// TIA Portal V20 export
FUNCTION_BLOCK "LER_RFID"   // FB115, LAD
// stored: Access Published, MemoryReserve 100, SetENOAutomatically false
   VAR_INPUT
      enable : Bool;
      enableManualCmds : Bool;
      bobinChuck : Bool;
   END_VAR
   VAR_OUTPUT
      error : Bool;
      status : DWord;
   END_VAR
   VAR_IN_OUT
      RFID_Chanel : TO_IDENT;
      IdentRfAntena : "LSicar_typeIdentInterfaceHmi";
      moduleInterface : "LER_typeRFIDInterface";
   END_VAR
   VAR
      instResetReader : Reset_Reader;
      instRead : Read;
      instWrite : Write;
      instInventory : Inventory;
      statResetReaderUDT : "LER_typeResetReaderUDT";
      statReadUDT : "LER_typeReadWriteUDT";
      statWriteUDT : "LER_typeReadWriteUDT";
      statInventoryUDT : "LER_typeInventoryUDT";
      statResultRFIDReset : Bool;
      statPulse : Array[0..9] of Bool;
      statTonTimer : TON_TIME;
      statBobinData : IID_IN_I_81;
      statRFID_str : String[32];
      statEPCID_str : String[32];
      statHi : Byte;
      statLo : Byte;
      statHexArray : Array[0..15] of Char;
   END_VAR
   VAR_TEMP
      resultRFID_Delete : String;
      resultData_Delete : WString;
      resultid_Delete : SInt;
      tempRet_Val : Word;
      tempBobinEPCData : Array[1..62] of Byte;
      i : Int;
      HI : Int;
      LO : Int;
   END_VAR
   VAR CONSTANT
      FALSE : Bool;
      deviceType : WString := WSTRING#'RF680R';
      deviceId : SInt := 6;   // RF600 = 6
      tagType : WString := WSTRING#'RFID';
   END_VAR
   // statHexArray[0] := '0';
   // statHexArray[1] := '1';
   // statHexArray[2] := '2';
   // statHexArray[3] := '3';
   // statHexArray[4] := '4';
   // statHexArray[5] := '5';
   // statHexArray[6] := '6';
   // statHexArray[7] := '7';
   // statHexArray[8] := '8';
   // statHexArray[9] := '9';
   // statHexArray[10] := 'A';
   // statHexArray[11] := 'B';
   // statHexArray[12] := 'C';
   // statHexArray[13] := 'D';
   // statHexArray[14] := 'E';
   // statHexArray[15] := 'F';
   VAR_TEMP   // added for the SCL form of the ladder/FBD networks
      _w1 : Bool;
   END_VAR
BEGIN

REGION Network 1 (SCL): Input Mapping
   // READ
   #statReadUDT.Input.addrTag := #moduleInterface.configuration.addrTag;
   #statReadUDT.Input.lengthData := #moduleInterface.configuration.lengthData;

   // INVENTORY
   #statInventoryUDT.Input.attribute := #moduleInterface.configuration.attribute;
   #statInventoryUDT.Input.duration := #moduleInterface.configuration.duration;
   #statInventoryUDT.Input.durUnit := #moduleInterface.configuration.durUnit;

   IF #enableManualCmds OR true THEN
       #statResetReaderUDT.Input.execute := #moduleInterface.commands.ResetReq OR #IdentRfAntena.pushbutton.%X0;
       #statReadUDT.Input.execute := #moduleInterface.commands.readReq OR #IdentRfAntena.pushbutton.%X1;
       #statWriteUDT.Input.execute := #moduleInterface.commands.writeReq OR #IdentRfAntena.pushbutton.%X2;
       #statResultRFIDReset := #moduleInterface.commands.resultRFIDReset OR #IdentRfAntena.pushbutton.%X3;
       #statInventoryUDT.Input.execute := #moduleInterface.commands.inventoryReq OR #statReadUDT.Output.done;

   END_IF;
END_REGION

REGION Network 2: Reset Reader
   // The Reset block sets the reader to a operational state. The Reset also acknowledges error conditions of the reader and resets a reader from a falty state to a OK-state.
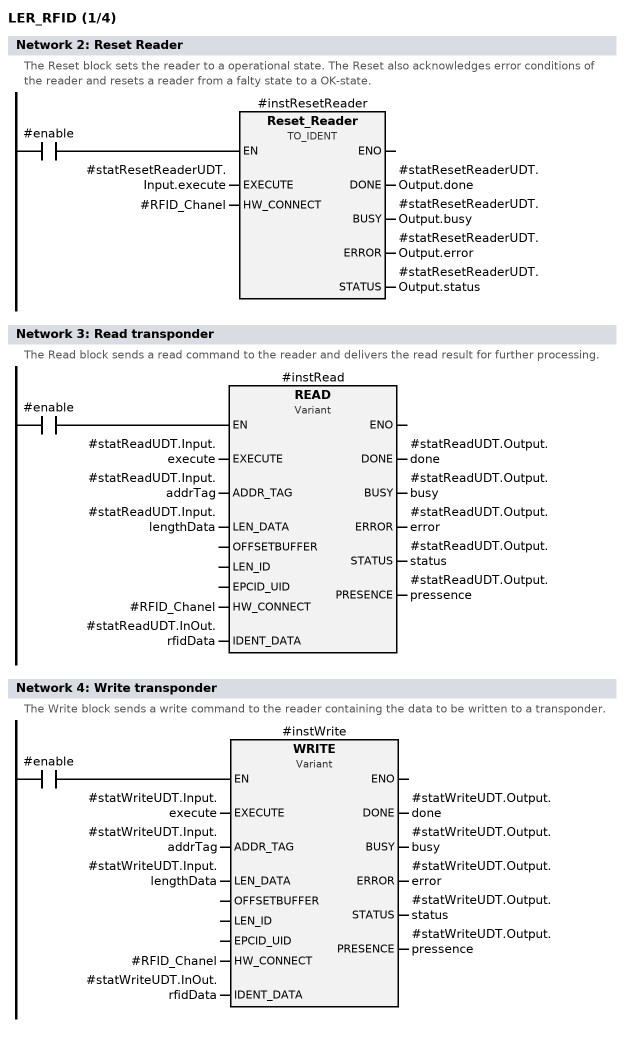
   RUNG wire#powerrail
      Contact( #enable )
      { S7_Templates := "connect_type := TO_IDENT" } #instResetReader.Reset_Reader(EXECUTE := #statResetReaderUDT.Input.execute, HW_CONNECT := #RFID_Chanel, DONE => #statResetReaderUDT.Output.done, BUSY => #statResetReaderUDT.Output.busy, ERROR => #statResetReaderUDT.Output.error, STATUS => #statResetReaderUDT.Output.status)
   END_RUNG
   // the same network as SCL:
   IF #enable THEN
       #instResetReader(EXECUTE := #statResetReaderUDT.Input.execute,   // Reset_Reader
                        HW_CONNECT := #RFID_Chanel,
                        DONE => #statResetReaderUDT.Output.done,
                        BUSY => #statResetReaderUDT.Output.busy,
                        ERROR => #statResetReaderUDT.Output.error,
                        STATUS => #statResetReaderUDT.Output.status);
   END_IF;
END_REGION

REGION Network 3: Read transponder
   // The Read block sends a read command to the reader and delivers the read result for further processing.
   RUNG wire#powerrail
      Contact( #enable )
      { S7_Templates := "[ident_data_type := Variant, connect_type := TO_IDENT]" } #instRead.Read(EXECUTE := #statReadUDT.Input.execute, ADDR_TAG := #statReadUDT.Input.addrTag, LEN_DATA := #statReadUDT.Input.lengthData, OFFSETBUFFER :=, LEN_ID :=, EPCID_UID :=, HW_CONNECT := #RFID_Chanel, IDENT_DATA := #statReadUDT.InOut.rfidData, DONE => #statReadUDT.Output.done, BUSY => #statReadUDT.Output.busy, ERROR => #statReadUDT.Output.error, STATUS => #statReadUDT.Output.status, PRESENCE => #statReadUDT.Output.pressence)
   END_RUNG
   // the same network as SCL:
   IF #enable THEN
       #instRead(EXECUTE := #statReadUDT.Input.execute,   // Read
                 ADDR_TAG := #statReadUDT.Input.addrTag,
                 LEN_DATA := #statReadUDT.Input.lengthData,
                 HW_CONNECT := #RFID_Chanel,
                 IDENT_DATA := #statReadUDT.InOut.rfidData,
                 DONE => #statReadUDT.Output.done,
                 BUSY => #statReadUDT.Output.busy,
                 ERROR => #statReadUDT.Output.error,
                 STATUS => #statReadUDT.Output.status,
                 PRESENCE => #statReadUDT.Output.pressence);
   END_IF;
END_REGION

REGION Network 4: Write transponder
   // The Write block sends a write command to the reader containing the data to be written to a transponder.
   RUNG wire#powerrail
      Contact( #enable )
      { S7_Templates := "[ident_data_type := Variant, connect_type := TO_IDENT]" } #instWrite.Write(EXECUTE := #statWriteUDT.Input.execute, ADDR_TAG := #statWriteUDT.Input.addrTag, LEN_DATA := #statWriteUDT.Input.lengthData, OFFSETBUFFER :=, LEN_ID :=, EPCID_UID :=, HW_CONNECT := #RFID_Chanel, IDENT_DATA := #statWriteUDT.InOut.rfidData, DONE => #statWriteUDT.Output.done, BUSY => #statWriteUDT.Output.busy, ERROR => #statWriteUDT.Output.error, STATUS => #statWriteUDT.Output.status, PRESENCE => #statWriteUDT.Output.pressence)
   END_RUNG
   // the same network as SCL:
   IF #enable THEN
       #instWrite(EXECUTE := #statWriteUDT.Input.execute,   // Write
                  ADDR_TAG := #statWriteUDT.Input.addrTag,
                  LEN_DATA := #statWriteUDT.Input.lengthData,
                  HW_CONNECT := #RFID_Chanel,
                  IDENT_DATA := #statWriteUDT.InOut.rfidData,
                  DONE => #statWriteUDT.Output.done,
                  BUSY => #statWriteUDT.Output.busy,
                  ERROR => #statWriteUDT.Output.error,
                  STATUS => #statWriteUDT.Output.status,
                  PRESENCE => #statWriteUDT.Output.pressence);
   END_IF;
END_REGION

REGION Network 5: Inventory
   // The Inventory block sends an inventory command to the reader and delivers the result for further processing
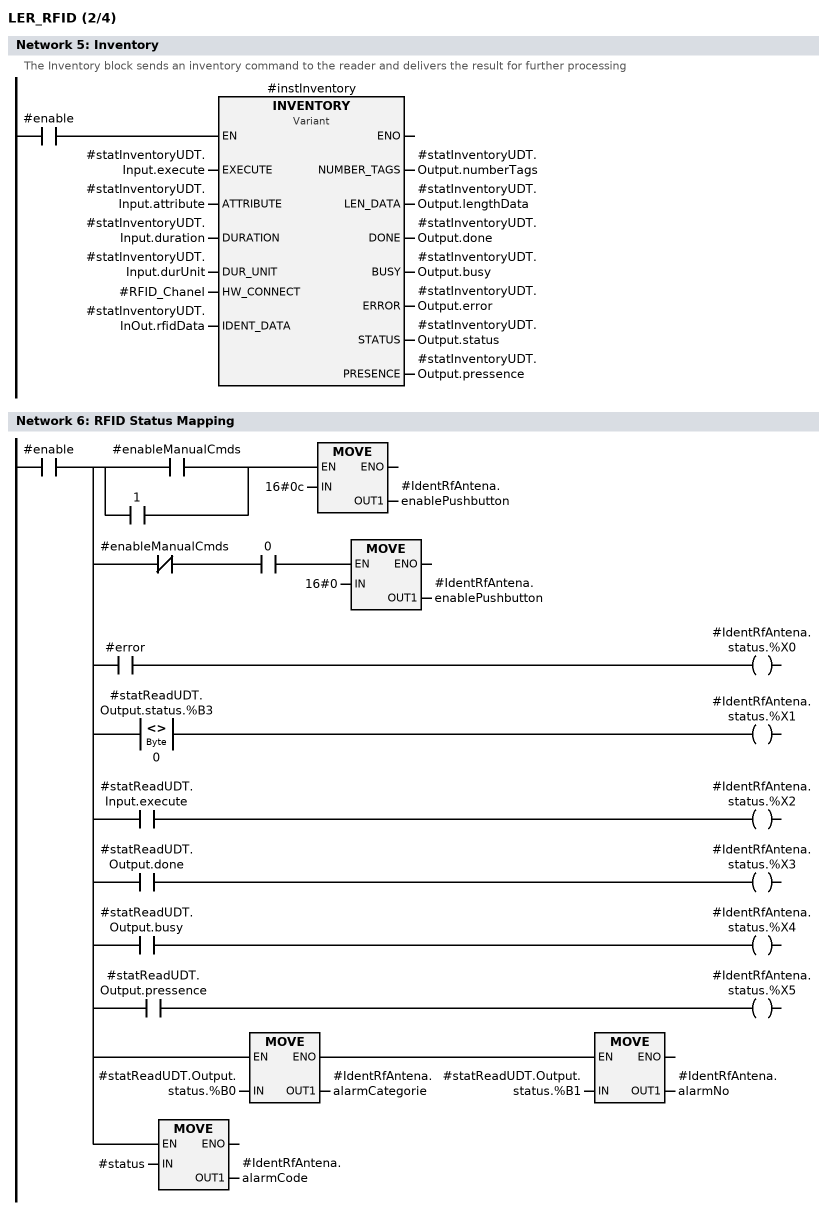
   RUNG wire#powerrail
      Contact( #enable )
      { S7_Templates := "[ident_data_type := Variant, connect_type := TO_IDENT]" } #instInventory.Inventory(EXECUTE := #statInventoryUDT.Input.execute, ATTRIBUTE := #statInventoryUDT.Input.attribute, DURATION := #statInventoryUDT.Input.duration, DUR_UNIT := #statInventoryUDT.Input.durUnit, HW_CONNECT := #RFID_Chanel, IDENT_DATA := #statInventoryUDT.InOut.rfidData, NUMBER_TAGS => #statInventoryUDT.Output.numberTags, LEN_DATA => #statInventoryUDT.Output.lengthData, DONE => #statInventoryUDT.Output.done, BUSY => #statInventoryUDT.Output.busy, ERROR => #statInventoryUDT.Output.error, STATUS => #statInventoryUDT.Output.status, PRESENCE => #statInventoryUDT.Output.pressence)
   END_RUNG
   // the same network as SCL:
   IF #enable THEN
       #instInventory(EXECUTE := #statInventoryUDT.Input.execute,   // Inventory
                      ATTRIBUTE := #statInventoryUDT.Input.attribute,
                      DURATION := #statInventoryUDT.Input.duration,
                      DUR_UNIT := #statInventoryUDT.Input.durUnit,
                      HW_CONNECT := #RFID_Chanel,
                      IDENT_DATA := #statInventoryUDT.InOut.rfidData,
                      NUMBER_TAGS => #statInventoryUDT.Output.numberTags,
                      LEN_DATA => #statInventoryUDT.Output.lengthData,
                      DONE => #statInventoryUDT.Output.done,
                      BUSY => #statInventoryUDT.Output.busy,
                      ERROR => #statInventoryUDT.Output.error,
                      STATUS => #statInventoryUDT.Output.status,
                      PRESENCE => #statInventoryUDT.Output.pressence);
   END_IF;
END_REGION

REGION Network 6: RFID Status Mapping
   RUNG wire#powerrail
      Contact( #enable )
      wire#w1
      Contact( #enableManualCmds )
      wire#w2
      Move(in := 16#0c, out1 => #IdentRfAntena.enablePushbutton)
   END_RUNG
   RUNG wire#w1
      Contact( 1 )
   END_RUNG wire#w2
   RUNG wire#w1
      I_Contact( #enableManualCmds )
      Contact( 0 )
      Move(in := 16#0, out1 => #IdentRfAntena.enablePushbutton)
   END_RUNG
   RUNG wire#w1
      Contact( #error )
      Coil( #IdentRfAntena.status.%X0 )
   END_RUNG
   RUNG wire#w1
      { S7_Templates := "SrcType := Byte" } NE_Contact(in1 := #statReadUDT.Output.status.%B3, in2 := 0)
      Coil( #IdentRfAntena.status.%X1 )
   END_RUNG
   RUNG wire#w1
      Contact( #statReadUDT.Input.execute )
      Coil( #IdentRfAntena.status.%X2 )
   END_RUNG
   RUNG wire#w1
      Contact( #statReadUDT.Output.done )
      Coil( #IdentRfAntena.status.%X3 )
   END_RUNG
   RUNG wire#w1
      Contact( #statReadUDT.Output.busy )
      Coil( #IdentRfAntena.status.%X4 )
   END_RUNG
   RUNG wire#w1
      Contact( #statReadUDT.Output.pressence )
      Coil( #IdentRfAntena.status.%X5 )
   END_RUNG
   RUNG wire#w1
      Move(in := #statReadUDT.Output.status.%B0, out1 => #IdentRfAntena.alarmCategorie)
      Move(in := #statReadUDT.Output.status.%B1, out1 => #IdentRfAntena.alarmNo)
   END_RUNG
   RUNG wire#w1
      Move(in := #status, out1 => #IdentRfAntena.alarmCode)
   END_RUNG
   // the same network as SCL:
   IF #enable AND (#enableManualCmds OR 1) THEN #IdentRfAntena.enablePushbutton := 16#0c; END_IF;
   IF #enable AND NOT #enableManualCmds AND 0 THEN #IdentRfAntena.enablePushbutton := 16#0; END_IF;
   #IdentRfAntena.status.%X0 := #enable AND #error;
   #IdentRfAntena.status.%X1 := #enable AND (#statReadUDT.Output.status.%B3 <> 0);
   #IdentRfAntena.status.%X2 := #enable AND #statReadUDT.Input.execute;
   #IdentRfAntena.status.%X3 := #enable AND #statReadUDT.Output.done;
   #IdentRfAntena.status.%X4 := #enable AND #statReadUDT.Output.busy;
   #IdentRfAntena.status.%X5 := #enable AND #statReadUDT.Output.pressence;
   IF #enable THEN
       #IdentRfAntena.alarmCategorie := #statReadUDT.Output.status.%B0;
       #IdentRfAntena.alarmNo := #statReadUDT.Output.status.%B1;
       #IdentRfAntena.alarmCode := #status;
   END_IF;
END_REGION

REGION Network 7 (SCL): RFID combination (Byte To string)
   IF #enable AND #statReadUDT.Output.done THEN
       #statRFID_str := '';

       FOR #i := 0 TO 15 DO
           #statHi := SHR(IN := #statReadUDT.InOut.rfidData[#i], N := 4);
           #statLo := #statReadUDT.InOut.rfidData[#i] AND 16#0F;
           #statRFID_str := CONCAT(IN1 := #statRFID_str, IN2 := #statHexArray[#statHi]);
           #statRFID_str := CONCAT(IN1 := #statRFID_str, IN2 := #statHexArray[#statLo]);
       END_FOR;
   END_IF;
END_REGION

REGION Network 8: RFID ID Sift
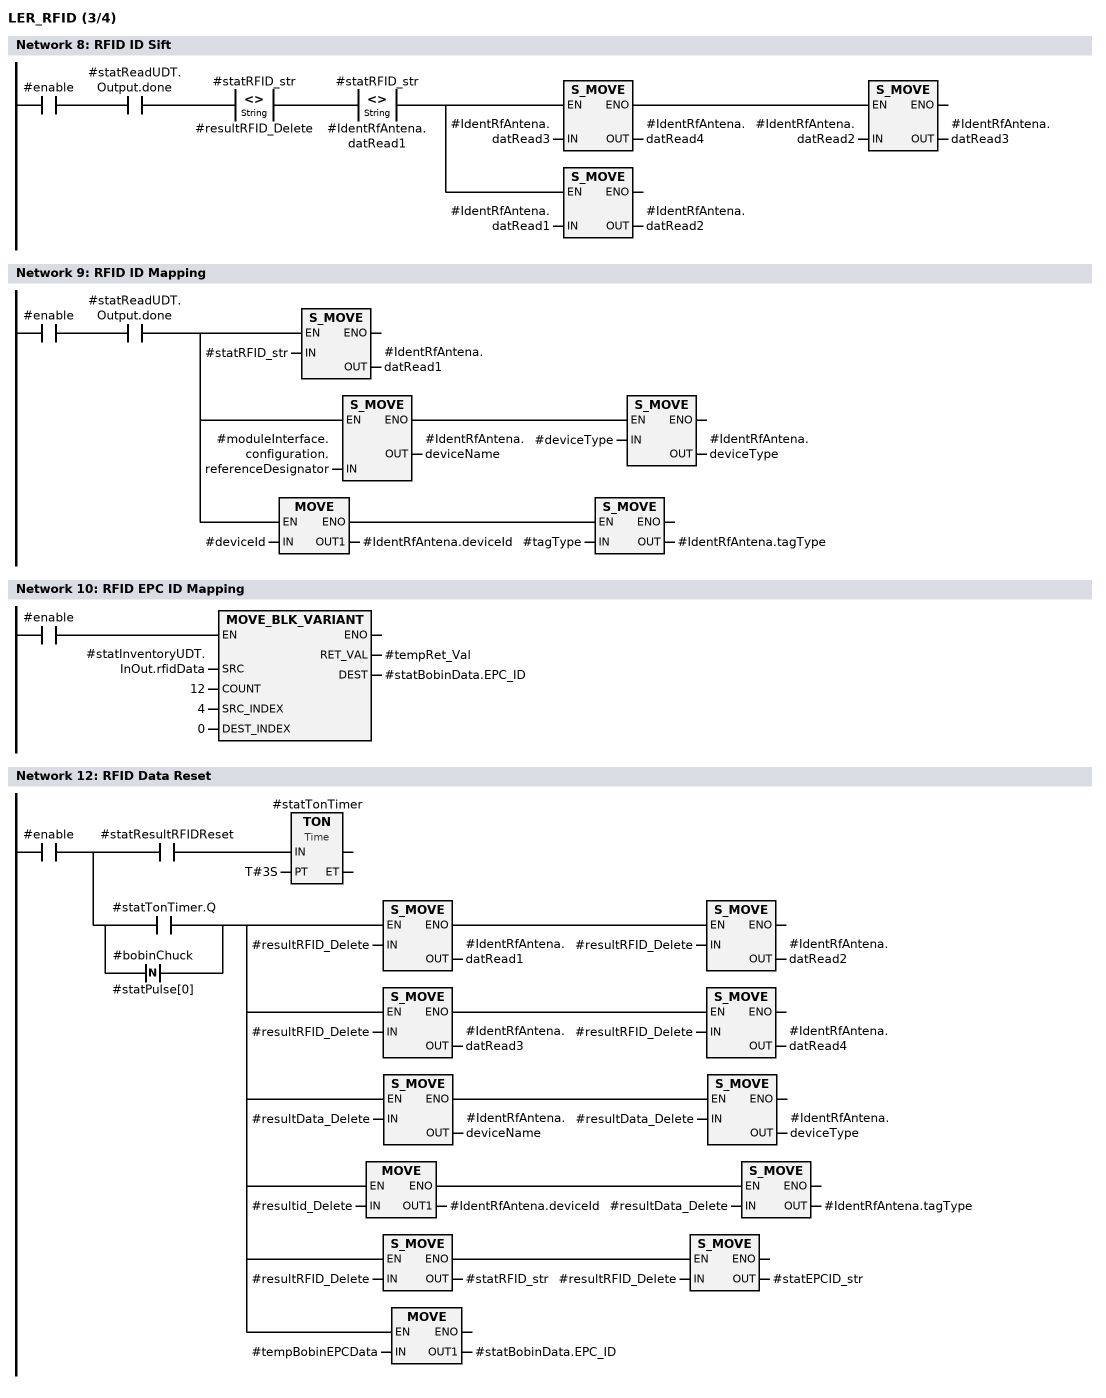
   RUNG wire#powerrail
      Contact( #enable )
      Contact( #statReadUDT.Output.done )
      { S7_Templates := "SrcType := String" } NE_Contact(in1 := #statRFID_str, in2 := #resultRFID_Delete)
      { S7_Templates := "SrcType := String" } NE_Contact(in1 := #statRFID_str, in2 := #IdentRfAntena.datRead1)
      wire#w1
      S_Move(in := #IdentRfAntena.datRead3, out => #IdentRfAntena.datRead4)
      S_Move(in := #IdentRfAntena.datRead2, out => #IdentRfAntena.datRead3)
   END_RUNG
   RUNG wire#w1
      S_Move(in := #IdentRfAntena.datRead1, out => #IdentRfAntena.datRead2)
   END_RUNG
   // the same network as SCL:
   IF #enable AND #statReadUDT.Output.done AND (#statRFID_str <> #resultRFID_Delete) AND (#statRFID_str <> #IdentRfAntena.datRead1) THEN
       #IdentRfAntena.datRead4 := #IdentRfAntena.datRead3;
       #IdentRfAntena.datRead3 := #IdentRfAntena.datRead2;
       #IdentRfAntena.datRead2 := #IdentRfAntena.datRead1;
   END_IF;
END_REGION

REGION Network 9: RFID ID Mapping
   RUNG wire#powerrail
      Contact( #enable )
      Contact( #statReadUDT.Output.done )
      wire#w1
      S_Move(in := #statRFID_str, out => #IdentRfAntena.datRead1)
   END_RUNG
   RUNG wire#w1
      S_Move(in := #moduleInterface.configuration.referenceDesignator, out => #IdentRfAntena.deviceName)
      S_Move(in := #deviceType, out => #IdentRfAntena.deviceType)
   END_RUNG
   RUNG wire#w1
      Move(in := #deviceId, out1 => #IdentRfAntena.deviceId)
      S_Move(in := #tagType, out => #IdentRfAntena.tagType)
   END_RUNG
   // the same network as SCL:
   IF #enable AND #statReadUDT.Output.done THEN
       #IdentRfAntena.datRead1 := #statRFID_str;
       #IdentRfAntena.deviceName := #moduleInterface.configuration.referenceDesignator;
       #IdentRfAntena.deviceType := #deviceType;
       #IdentRfAntena.deviceId := #deviceId;
       #IdentRfAntena.tagType := #tagType;
   END_IF;
END_REGION

REGION Network 10: RFID EPC ID Mapping
   RUNG wire#powerrail
      Contact( #enable )
      MOVE_BLK_VARIANT(SRC := #statInventoryUDT.InOut.rfidData, COUNT := 12, SRC_INDEX := 4, DEST_INDEX := 0, Ret_Val => #tempRet_Val, DEST => #statBobinData.EPC_ID)
   END_RUNG
   // the same network as SCL:
   IF #enable THEN
       #tempRet_Val := MOVE_BLK_VARIANT(SRC := #statInventoryUDT.InOut.rfidData,
                               COUNT := 12,
                               SRC_INDEX := 4,
                               DEST_INDEX := 0,
                               DEST => #statBobinData.EPC_ID);
   END_IF;
END_REGION

REGION Network 11 (SCL): RFID EPC ID Combination (Byte To string)
   IF #enable AND #statInventoryUDT.Output.done THEN
       #statEPCID_str := '';

       FOR #i := 1 TO 12 DO
           #statHi := SHR(IN := #statBobinData.EPC_ID[#i], N := 4);
           #statLo := #statBobinData.EPC_ID[#i] AND 16#0F;
           #statEPCID_str := CONCAT(IN1 := #statEPCID_str, IN2 := #statHexArray[#statHi]);
           #statEPCID_str := CONCAT(IN1 := #statEPCID_str, IN2 := #statHexArray[#statLo]);
       END_FOR;
   END_IF;
END_REGION

REGION Network 12: RFID Data Reset
   RUNG wire#powerrail
      Contact( #enable )
      wire#w1
      Contact( #statResultRFIDReset )
      { S7_Templates := "time_type := Time" } #statTonTimer.TON(pt := T#3S, et =>)
   END_RUNG
   RUNG wire#w1
      Contact( #statTonTimer.Q )
      wire#w2
      S_Move(in := #resultRFID_Delete, out => #IdentRfAntena.datRead1)
      S_Move(in := #resultRFID_Delete, out => #IdentRfAntena.datRead2)
   END_RUNG
   RUNG wire#w1
      N_Contact(operand := #bobinChuck, bit := #statPulse[0])
   END_RUNG wire#w2
   RUNG wire#w2
      S_Move(in := #resultRFID_Delete, out => #IdentRfAntena.datRead3)
      S_Move(in := #resultRFID_Delete, out => #IdentRfAntena.datRead4)
   END_RUNG
   RUNG wire#w2
      S_Move(in := #resultData_Delete, out => #IdentRfAntena.deviceName)
      S_Move(in := #resultData_Delete, out => #IdentRfAntena.deviceType)
   END_RUNG
   RUNG wire#w2
      Move(in := #resultid_Delete, out1 => #IdentRfAntena.deviceId)
      S_Move(in := #resultData_Delete, out => #IdentRfAntena.tagType)
   END_RUNG
   RUNG wire#w2
      S_Move(in := #resultRFID_Delete, out => #statRFID_str)
      S_Move(in := #resultRFID_Delete, out => #statEPCID_str)
   END_RUNG
   RUNG wire#w2
      Move(in := #tempBobinEPCData, out1 => #statBobinData.EPC_ID)
   END_RUNG
   // the same network as SCL:
   #statTonTimer(IN := #enable AND #statResultRFIDReset, PT := T#3S);   // TON
   #_w1 := #enable AND NOT #bobinChuck AND #statPulse[0];   // falling edge of #bobinChuck
   #statPulse[0] := #bobinChuck;
   IF (#enable AND #statTonTimer.Q) OR #_w1 THEN
       #IdentRfAntena.datRead1 := #resultRFID_Delete;
       #IdentRfAntena.datRead2 := #resultRFID_Delete;
       #IdentRfAntena.datRead3 := #resultRFID_Delete;
       #IdentRfAntena.datRead4 := #resultRFID_Delete;
       #IdentRfAntena.deviceName := #resultData_Delete;
       #IdentRfAntena.deviceType := #resultData_Delete;
       #IdentRfAntena.deviceId := #resultid_Delete;
       #IdentRfAntena.tagType := #resultData_Delete;
       #statRFID_str := #resultRFID_Delete;
       #statEPCID_str := #resultRFID_Delete;
       #statBobinData.EPC_ID := #tempBobinEPCData;
   END_IF;
END_REGION

REGION Network 13: Error Check
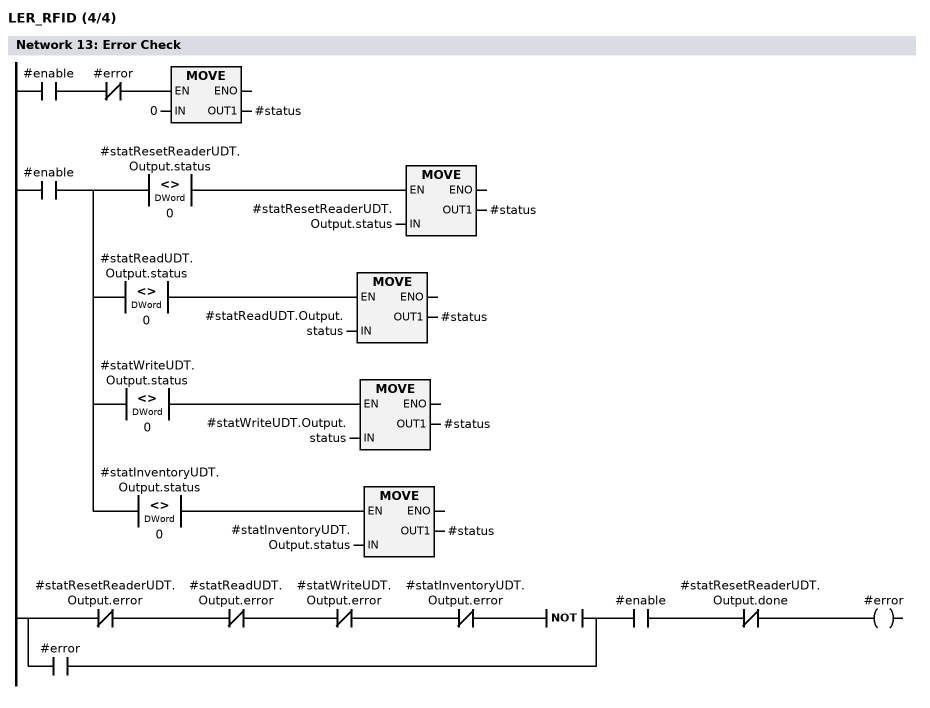
   RUNG wire#powerrail
      Contact( #enable )
      I_Contact( #error )
      Move(in := 0, out1 => #status)
   END_RUNG
   RUNG wire#powerrail
      Contact( #enable )
      wire#w1
      { S7_Templates := "SrcType := DWord" } NE_Contact(in1 := #statResetReaderUDT.Output.status, in2 := 0)
      Move(in := #statResetReaderUDT.Output.status, out1 => #status)
   END_RUNG
   RUNG wire#w1
      { S7_Templates := "SrcType := DWord" } NE_Contact(in1 := #statReadUDT.Output.status, in2 := 0)
      Move(in := #statReadUDT.Output.status, out1 => #status)
   END_RUNG
   RUNG wire#w1
      { S7_Templates := "SrcType := DWord" } NE_Contact(in1 := #statWriteUDT.Output.status, in2 := 0)
      Move(in := #statWriteUDT.Output.status, out1 => #status)
   END_RUNG
   RUNG wire#w1
      { S7_Templates := "SrcType := DWord" } NE_Contact(in1 := #statInventoryUDT.Output.status, in2 := 0)
      Move(in := #statInventoryUDT.Output.status, out1 => #status)
   END_RUNG
   RUNG wire#powerrail
      I_Contact( #statResetReaderUDT.Output.error )
      I_Contact( #statReadUDT.Output.error )
      I_Contact( #statWriteUDT.Output.error )
      I_Contact( #statInventoryUDT.Output.error )
      Not()
      wire#w2
      Contact( #enable )
      I_Contact( #statResetReaderUDT.Output.done )
      Coil( #error )
   END_RUNG
   RUNG wire#powerrail
      Contact( #error )
   END_RUNG wire#w2
   // the same network as SCL:
   IF #enable AND NOT #error THEN #status := 0; END_IF;
   IF #enable AND (#statResetReaderUDT.Output.status <> 0) THEN
       #status := #statResetReaderUDT.Output.status;
   END_IF;
   IF #enable AND (#statReadUDT.Output.status <> 0) THEN #status := #statReadUDT.Output.status; END_IF;
   IF #enable AND (#statWriteUDT.Output.status <> 0) THEN #status := #statWriteUDT.Output.status; END_IF;
   IF #enable AND (#statInventoryUDT.Output.status <> 0) THEN
       #status := #statInventoryUDT.Output.status;
   END_IF;
   #error := (NOT (NOT #statResetReaderUDT.Output.error AND NOT #statReadUDT.Output.error AND NOT #statWriteUDT.Output.error AND NOT #statInventoryUDT.Output.error) OR #error) AND #enable AND NOT #statResetReaderUDT.Output.done;
END_REGION

REGION Network 14 (SCL): Output Mapping
   #moduleInterface.monitoring.ResultData := #IdentRfAntena;
   #moduleInterface.monitoring.error := #error;
   #moduleInterface.monitoring.status:= #status;
END_REGION
END_FUNCTION_BLOCK
